{attribute 'linkalways'} 
{attribute 'no_explicit_call' := 'This FB is a CLASS and must be accessed using methods or properties'}
{attribute 'enable_dynamic_creation'}
FUNCTION_BLOCK FINAL TAN_LREAL EXTENDS Node
VAR
	in : _LREAL(0.0);
	out : _LREAL(0.0);
END_VAR

METHOD PUBLIC Clone : I_Node
VAR
	pNode : POINTER TO TAN_LREAL;
END_VAR
pNode := __NEW(TAN_LREAL);
Clone := pNode^;
END_METHOD

METHOD FB_init : BOOL
VAR_INPUT
	bInitRetains : BOOL; // if TRUE, the retain variables are initialized (warm start / cold start)
	bInCopyCode : BOOL;  // if TRUE, the instance afterwards gets moved into the copy code (online change)
END_VAR
AddInput('in',THIS^.in);
AddOutput('out', THIS^.out);
END_METHOD

METHOD PROTECTED OnExecute
VAR
END_VAR
out.Value := TAN(in.Value);
END_METHOD

END_FUNCTION_BLOCK

(* stored: Version 1.1.0.1, ProductVersion 3.1.4024.15
   POU TAN_LREAL: Id {dc172830-627f-42f0-8201-6788d2fcacbd}, SpecialFunc None
   Folder Constructor: Id {15a99db1-bbc1-4880-ac0e-53b32f3658f2}
   Method Clone: Id {446f715b-9c3e-400b-83b9-427b406773d5}
   Method FB_init: Id {bda5aceb-d68d-4107-a833-dda49e79df5f}
   Method OnExecute: Id {3dc61542-1023-4e40-9c54-9251fc62e5e9} *)
